{attribute 'qualified_only'}
{attribute 'strict'}

//-----------------------------------------------------------------------------------------
//
//                  				ENUM_Door
//
//						Enumération des types de porte(s)			
//-----------------------------------------------------------------------------------------
//
//Auteur: G.GOETZ
//Création: 13.01.2026
//Dernière modification : 13.01.2026 (G.GOETZ)
//       			
//-----------------------------------------------------------------------------------------
//
//     							Liste des modifications  	
//
// 13.01.2026 (G.GOETZ) -> Création		
//-----------------------------------------------------------------------------------------

TYPE ENUM_Position_Magazine :
(
	Unknow := 0 , // Unknow position
	Top := 1 , // At the top of the Magazine
	Bottom := 2 // At the bootom of the Magazine 
);
END_TYPE

(* stored: Version 1.1.0.1, ProductVersion 3.1.4024.13
   DUT ENUM_Position_Magazine: Id {ffaa26ba-7347-4a8b-bd50-1dba5fe66683} *)
